# EPICS substitutions: iocs/MC07/tpmacApp/Db/pmac_physical_limit.substitutions
file "${TOP}/db/pmac_physical_limit.db"
{
pattern
{SYS,            DEV,                    }
{"XF:06BMA-BI",  "{XAFS-Ax:Tbl_YU}"      }
{"XF:06BMA-BI",  "{XAFS-Ax:Tbl_YDO}"     }
{"XF:06BMA-BI",  "{XAFS-Ax:Tbl_YDI}"     }
{"XF:06BMA-BI",  "{XAFS-Ax:Tbl_XU}"      }
{"XF:06BMA-BI",  "{XAFS-Ax:Tbl_XD}"      }
{"XF:06BMA-BI",  "{XAFS-Ax:RotH}"        }
{"XF:06BMA-BI",  "{XAFS-Ax:RotB}"        }
{"XF:06BMA-BI",  "{XAFS-Ax:RotS}"        }
}
